FUNCTION_BLOCK FB_TouchProbe EXTENDS FB_Xfc
VAR
  _Ctrl             : REFERENCE TO ARRAY[1..MAX_TOUCH_PROBE] OF ST_CTRL_TOUCH_PROBE;
  _State            : REFERENCE TO ARRAY[1..MAX_TOUCH_PROBE] OF ST_STATE_TOUCH_PROBE;

  _Input            : POINTER TO ARRAY[1..MAX_TOUCH_PROBE] OF ST_MTI_Input;
  _InputState       : POINTER TO ARRAY[1..MAX_TOUCH_PROBE] OF ST_MTI_STATUS;

  _Index            : UDINT;
  _AxisId           : UDINT;
  _AxisIndex        : UDINT;

  _CtrlLocal        : ST_CTRL_TOUCH_PROBE;  // control data is copied to local on start of function
  _McDirection      : Tc2_MC2.MC_Direction;

  _eStateProgress   : E_PROGRESS;
  _eResult          : E_PROGRESS;

  _rtrigEnable      : Tc2_Standard.R_TRIG;
  _TrigCount        : UDINT;

  _CurrentTime      : ULINT;
  _CurrentTimeShort : UDINT;
  _LatchTime        : UDINT;
  _LatchState       : Bool;

  _bError           : BOOL;
  _stMsg            : ST_Message;
  _MessageLevel     : E_MessageType;
END_VAR

PROPERTY Ctrl : REFERENCE TO ARRAY [1..MAX_TOUCH_PROBE] OF ST_CTRL_TOUCH_PROBE
SET
_Ctrl REF= Ctrl;
END_SET
END_PROPERTY

METHOD Cycle : BOOL
VAR_INPUT
END_VAR
//-----------------------------------------------------------------------------
//-----------------------------------------------------------------------------
//  Check Enable
//-----------------------------------------------------------------------------
IF NOT _Ctrl[_Index].Enable
THEN
  // clear function state if not enabled
  _eStateProgress                   := E_PROGRESS.PROGRESS_INVALID;
  _LatchState                       := FALSE;
  _State[_Index].State              := TO_UINT(_eStateProgress);
END_IF
//-----------------------------------------------------------------------------
//-----------------------------------------------------------------------------
//  set message device
//-----------------------------------------------------------------------------
_eDeviceFunction                    := e_Device.XfcTouchProbe + _Index;
//-----------------------------------------------------------------------------
//-----------------------------------------------------------------------------
//  rising trigger react to enable command
//-----------------------------------------------------------------------------
_rtrigEnable(CLK                    := _Ctrl[_Index].Enable);
//-----------------------------------------------------------------------------
//-----------------------------------------------------------------------------
//  main state machine
//-----------------------------------------------------------------------------
CASE _eStateProgress
OF
  E_PROGRESS.PROGRESS_INVALID:      // check input data
    IF _rtrigEnable.Q
    THEN
      _State[_Index].State          := TO_UINT(E_PROGRESS.PROGRESS_BUSY);
      _State[_Index].LatchPositive  := 0.0;
      _State[_Index].LatchNegative  := 0.0;

      _bError                       := FALSE;
      _eStateProgress               := E_PROGRESS.PROGRESS_INIT;

      _CtrlLocal                    := _Ctrl[_Index];   // copy control data to local, you may write new data onto struct as long as .Enable stays TRUE
      _CurrentTime                  := Tc2_EtherCAT.F_GetCurDcTickTime64();
      _CurrentTimeShort             := TO_UDINT(_CurrentTime AND 16#FFFFFFFF);

      _AxisId                       := _CtrlLocal.AxisId;   // TwinCAT NC AxisId
      _AxisIndex                    := GetIndex(_AxisId);   // corresponding index in axis array

      _stMsg.iErrorNumber           := 0;

      IF NOT (_AxisIndex > 0) OR NOT (_AxisId > 0)
      THEN
        _bError                     := TRUE;
        _stMsg.iErrorNumber         := 1;
        _stMsg.sText                := 'AxisId Invalid ';
        _eStateProgress             := E_PROGRESS.PROGRESS_STILL_WORKING;
      END_IF

      IF NOT (_CtrlLocal.Direction = MC_Positive_Direction) OR 
         NOT (_CtrlLocal.Direction = MC_Negative_Direction)
      THEN
        _bError                     := TRUE;
        _stMsg.iErrorNumber         := 2;
        _stMsg.sText                := 'Direction Invalid ';
        _eStateProgress             := E_PROGRESS.PROGRESS_STILL_WORKING;
      END_IF

      IF NOT IsFinite(F_LReal(_CtrlLocal.PositionStart))
      THEN
        _bError                     := TRUE;
        _stMsg.iErrorNumber         := 3;
        _stMsg.sText                := 'PositionStart not finite ';
        _eStateProgress             := E_PROGRESS.PROGRESS_STILL_WORKING;
      END_IF

      IF NOT IsFinite(F_LReal(_CtrlLocal.PositionEnd))
      THEN
        _bError                     := TRUE;
        _stMsg.iErrorNumber         := 4;
        _stMsg.sText                := 'PositionEnd not finite ';
        _eStateProgress             := E_PROGRESS.PROGRESS_STILL_WORKING;
      END_IF
    END_IF

  E_PROGRESS.PROGRESS_INIT:
      _eDeviceAxis                  := e_Device.XfcAxis + (_CtrlLocal.AxisId);
      _eStateProgress               := E_PROGRESS.PROGRESS_BUSY;

      IF (_MessageLevel = E_MessageType.eMessageVerbose)
      THEN
        _stMsg.eType                := E_MessageType.eMessageVerbose;
        _stMsg.eDevice              := _eDeviceFunction;
        _stMsg.eSubdevice           := e_Subdevice.XfcTouchProbe;
        _stMsg.iErrorNumber         := _eDeviceAxis;
        _stMsg.sText                := concat(TO_STRING(_eStateProgress), ': ');
        _stMsg.sText                := concat(_stMsg.sText, TO_STRING(e_Device.XfcAxis));
        _stMsg.sText                := concat(_stMsg.sText, '_ID_');
        _stMsg.sText                := concat(_stMsg.sText, TO_STRING(_AxisId));

        f_MessageSet(_stMsg);
      END_IF
END_CASE
//-----------------------------------------------------------------------------
//-----------------------------------------------------------------------------
CASE _eStateProgress
OF
  E_PROGRESS.PROGRESS_BUSY:
    _McDirection                    := _CtrlLocal.Direction;
    CASE _McDirection
    OF
      MC_Positive_Direction:
        IF (_ItfAxis[_AxisIndex].Position >= _CtrlLocal.PositionStart)
        THEN
          _eResult                  := PositionAtTime(FALSE, _CtrlLocal.AxisId, 0, _MessageLevel);
          _eStateProgress           := E_PROGRESS.PROGRESS_PREPARE;
        END_IF

      MC_Negative_Direction:
        IF (_ItfAxis[_AxisIndex].Position <= _CtrlLocal.PositionStart)
        THEN
          _eResult                  := PositionAtTime(FALSE, _CtrlLocal.AxisId, 0, _MessageLevel);
          _eStateProgress           := E_PROGRESS.PROGRESS_PREPARE;
        END_IF
    END_CASE
END_CASE
//-----------------------------------------------------------------------------
//-----------------------------------------------------------------------------
CASE _eStateProgress
OF
  E_PROGRESS.PROGRESS_PREPARE:
    CASE _McDirection
    OF
      MC_Positive_Direction:
        IF (_ItfAxis[_AxisIndex].Position > _CtrlLocal.PositionEnd)
        THEN
          _bError                   := TRUE;
          _stMsg.iErrorNumber       := 5;
          _stMsg.sText              := 'PositionEnd reached, no rising trigger ';
          _eStateProgress           := E_PROGRESS.PROGRESS_STILL_WORKING;
    
        ELSIF (_Input^[_Index].EventState) OR
              (_Input^[_Index].EventTime > _CurrentTimeShort)
        THEN
          _LatchState               := _Input^[_Index].EventState;
          _LatchTime                := _Input^[_Index].EventTime;
    
          IF (_MessageLevel = E_MessageType.eMessageVerbose)
          THEN
            _stMsg.eType            := E_MessageType.eMessageVerbose;
            _stMsg.eDevice          := _eDeviceFunction;
            _stMsg.eSubdevice       := e_Subdevice.XfcTouchProbe;
            _stMsg.iErrorNumber     := _LatchTime;
            _stMsg.sText            := concat(TO_STRING(_eStateProgress), ': ');
            _stMsg.sText            := concat(_stMsg.sText, TO_STRING(e_Device.XfcAxis));
    
            f_MessageSet(_stMsg);
          END_IF
          _eStateProgress           := E_PROGRESS.PROGRESS_STARTUP;
        END_IF

      MC_Negative_Direction:
        IF (_ItfAxis[_AxisIndex].Position < _CtrlLocal.PositionEnd)
        THEN
          _bError                   := TRUE;
          _stMsg.iErrorNumber       := 5;
          _stMsg.sText              := 'PositionEnd reached, no rising trigger ';
          _eStateProgress           := E_PROGRESS.PROGRESS_STILL_WORKING;
    
        ELSIF (_Input^[_Index].EventState) OR
              (_Input^[_Index].EventTime > _CurrentTimeShort)
        THEN
          _LatchState               := _Input^[_Index].EventState;
          _LatchTime                := _Input^[_Index].EventTime;
    
          IF (_MessageLevel = E_MessageType.eMessageVerbose)
          THEN
            _stMsg.eType            := E_MessageType.eMessageVerbose;
            _stMsg.eDevice          := _eDeviceFunction;
            _stMsg.eSubdevice       := e_Subdevice.XfcTouchProbe;
            _stMsg.iErrorNumber     := _LatchTime;
            _stMsg.sText            := concat(TO_STRING(_eStateProgress), ': ');
            _stMsg.sText            := concat(_stMsg.sText, TO_STRING(e_Device.XfcAxis));
    
            f_MessageSet(_stMsg);
          END_IF
          _eStateProgress           := E_PROGRESS.PROGRESS_STARTUP;
        END_IF
    END_CASE
END_CASE
//-----------------------------------------------------------------------------
//-----------------------------------------------------------------------------
CASE _eStateProgress
OF
  E_PROGRESS.PROGRESS_STARTUP:
    _eResult                        := PositionAtTime(TRUE, _CtrlLocal.AxisId, _LatchTime, _MessageLevel);

    IF (_eResult = E_PROGRESS.PROGRESS_ERROR)
    THEN
      _bError                       := TRUE;
      _stMsg.iErrorNumber           := 7;
      _stMsg.sText                  := 'PositionAtTime LatchPositive ';
      _eStateProgress               := E_PROGRESS.PROGRESS_STILL_WORKING;
      _eResult                      := PositionAtTime(FALSE, _CtrlLocal.AxisId, 0, _MessageLevel);

    ELSIF (_eResult = E_PROGRESS.PROGRESS_DONE)
    THEN
      _State[_Index].LatchPositive  := _XfcRecordedPosition[_AxisIndex];

      _CurrentTime                  := Tc2_EtherCAT.F_GetCurDcTickTime64();
      _CurrentTimeShort             := TO_UDINT(_CurrentTime AND 16#FFFFFFFF);

      IF (_MessageLevel = E_MessageType.eMessageVerbose)
      THEN
        _stMsg.eType                := E_MessageType.eMessageVerbose;
        _stMsg.eDevice              := _eDeviceFunction;
        _stMsg.eSubdevice           := e_Subdevice.XfcTouchProbe;
        _stMsg.iErrorNumber         := _LatchTime;
        _stMsg.sText                := concat(TO_STRING(_eStateProgress), ': ');
        _stMsg.sText                := concat(_stMsg.sText, TO_STRING(_XfcRecordedPosition[_AxisIndex]));

        f_MessageSet(_stMsg);
      END_IF
      _eStateProgress               := E_PROGRESS.PROGRESS_CHECK;
      _eResult                      := PositionAtTime(FALSE, _CtrlLocal.AxisId, 0, _MessageLevel);
    END_IF
END_CASE
//-----------------------------------------------------------------------------
//-----------------------------------------------------------------------------
CASE _eStateProgress
OF
  E_PROGRESS.PROGRESS_CHECK:
    CASE _McDirection
    OF
      MC_Positive_Direction:
        IF (_ItfAxis[_AxisIndex].Position > _CtrlLocal.PositionEnd)
        THEN
          _bError                   := TRUE;
          _stMsg.iErrorNumber       := 6;
          _stMsg.sText              := concat('PositionEnd reached, no falling trigger :', TO_STRING(_ItfAxis[_AxisIndex].Position));
          _eStateProgress           := E_PROGRESS.PROGRESS_STILL_WORKING;
    
        ELSIF NOT (_Input^[_Index].EventState) OR
              (_Input^[_Index].EventTime > _LatchTime - 1_000)
        THEN
          _LatchState               := _Input^[_Index].EventState;
          _LatchTime                := _Input^[_Index].EventTime;
    
          IF (_MessageLevel = E_MessageType.eMessageVerbose)
          THEN
            _stMsg.eType            := E_MessageType.eMessageVerbose;
            _stMsg.eDevice          := _eDeviceFunction;
            _stMsg.eSubdevice       := e_Subdevice.XfcTouchProbe;
            _stMsg.iErrorNumber     := _LatchTime;
            _stMsg.sText            := concat(TO_STRING(_eStateProgress), ': ');
            _stMsg.sText            := concat(_stMsg.sText, TO_STRING(e_Device.XfcAxis));
    
            f_MessageSet(_stMsg);
          END_IF
          _eStateProgress           := E_PROGRESS.PROGRESS_OCCUPIED;
        END_IF

      MC_Negative_Direction:
        IF (_ItfAxis[_AxisIndex].Position < _CtrlLocal.PositionEnd)
        THEN
          _bError                   := TRUE;
          _stMsg.iErrorNumber       := 6;
          _stMsg.sText              := concat('PositionEnd reached, no falling trigger :', TO_STRING(_ItfAxis[_AxisIndex].Position));
          _eStateProgress           := E_PROGRESS.PROGRESS_STILL_WORKING;
    
        ELSIF NOT (_Input^[_Index].EventState) OR
              (_Input^[_Index].EventTime > _LatchTime - 1_000)
        THEN
          _LatchState               := _Input^[_Index].EventState;
          _LatchTime                := _Input^[_Index].EventTime;
    
          IF (_MessageLevel = E_MessageType.eMessageVerbose)
          THEN
            _stMsg.eType            := E_MessageType.eMessageVerbose;
            _stMsg.eDevice          := _eDeviceFunction;
            _stMsg.eSubdevice       := e_Subdevice.XfcTouchProbe;
            _stMsg.iErrorNumber     := _LatchTime;
            _stMsg.sText            := concat(TO_STRING(_eStateProgress), ': ');
            _stMsg.sText            := concat(_stMsg.sText, TO_STRING(e_Device.XfcAxis));
    
            f_MessageSet(_stMsg);
          END_IF
          _eStateProgress           := E_PROGRESS.PROGRESS_OCCUPIED;
        END_IF
    END_CASE
END_CASE
//-----------------------------------------------------------------------------
//-----------------------------------------------------------------------------
CASE _eStateProgress
OF
  E_PROGRESS.PROGRESS_OCCUPIED:
    _eResult                        := PositionAtTime(TRUE, _CtrlLocal.AxisId, _LatchTime, _MessageLevel);

    IF (_eResult = E_PROGRESS.PROGRESS_ERROR)
    THEN
      _bError                       := TRUE;
      _stMsg.iErrorNumber           := 8;
      _stMsg.sText                  := 'PositionAtTime LatchNegative: ';
      _eStateProgress               := E_PROGRESS.PROGRESS_STILL_WORKING;
      _eResult                      := PositionAtTime(FALSE, _CtrlLocal.AxisId, 0, _MessageLevel);

    ELSIF (_eResult = E_PROGRESS.PROGRESS_DONE)
    THEN
      _State[_Index].LatchNegative  := _XfcRecordedPosition[_AxisIndex];

      IF (_MessageLevel = E_MessageType.eMessageVerbose)
      THEN
        _stMsg.eType                := E_MessageType.eMessageVerbose;
        _stMsg.eDevice              := _eDeviceFunction;
        _stMsg.eSubdevice           := e_Subdevice.XfcTouchProbe;
        _stMsg.iErrorNumber         := _LatchTime;
        _stMsg.sText                := concat(TO_STRING(_eStateProgress), ': ');
        _stMsg.sText                := concat(_stMsg.sText, TO_STRING(_XfcRecordedPosition[_AxisIndex]));

        f_MessageSet(_stMsg);
      END_IF
      _eStateProgress               := E_PROGRESS.PROGRESS_WORKING;
      _eResult                      := PositionAtTime(FALSE, _CtrlLocal.AxisId, 0, _MessageLevel);
    END_IF
END_CASE
//-----------------------------------------------------------------------------
//-----------------------------------------------------------------------------
CASE _eStateProgress
OF
  E_PROGRESS.PROGRESS_WORKING:
    _eStateProgress                 := E_PROGRESS.PROGRESS_STILL_WORKING;
END_CASE
//-----------------------------------------------------------------------------
//-----------------------------------------------------------------------------
CASE _eStateProgress
OF
  E_PROGRESS.PROGRESS_STILL_WORKING:
    IF NOT _bError
    THEN
      _eStateProgress               := E_PROGRESS.PROGRESS_DONE;

      IF (_MessageLevel > E_MessageType.eMessageWarning)
      THEN
        _stMsg.eType                := E_MessageType.eMessageInfo;
        _stMsg.eDevice              := _eDeviceFunction;
        _stMsg.eSubdevice           := e_Subdevice.XfcTouchProbe;
        _stMsg.iErrorNumber         := _eDeviceAxis;
        _stMsg.sText                := concat(TO_STRING(_eStateProgress), ': ');
        _stMsg.sText                := concat(_stMsg.sText, TO_STRING(e_Device.XfcAxis));
        _stMsg.sText                := concat(_stMsg.sText, '_ID_');
        _stMsg.sText                := concat(_stMsg.sText, TO_STRING(_AxisId));

        f_MessageSet(_stMsg);
      END_IF
      _State[_Index].State          := TO_UINT(_eStateProgress);
    ELSE
      _eStateProgress               := E_PROGRESS.PROGRESS_ERROR;

      _stMsg.eType                  := E_MessageType.eMessageError;
      _stMsg.eDevice                := _eDeviceFunction;
      _stMsg.eSubdevice             := e_Subdevice.XfcTouchProbe;
      _stMsg.sText                  := concat(_stMsg.sText, TO_STRING(_eStateProgress));
      _stMsg.sText                  := concat(_stMsg.sText, ': ');
      _stMsg.sText                  := concat(_stMsg.sText, TO_STRING(e_Device.XfcAxis));
      _stMsg.sText                  := concat(_stMsg.sText, '_ID_');
      _stMsg.sText                  := concat(_stMsg.sText, TO_STRING(_AxisId));

      f_MessageSet(_stMsg);
      _State[_Index].State          := TO_UINT(_eStateProgress) + TO_UINT(_stMsg.iErrorNumber);
    END_IF
END_CASE
END_METHOD

PROPERTY Index : udint
GET
Index := _Index;
END_GET
SET
_Index := Index;
END_SET
END_PROPERTY

PROPERTY Input : pointer TO ARRAY [1..MAX_TOUCH_PROBE] OF ST_MTI_Input
SET
_Input := Input;
END_SET
END_PROPERTY

PROPERTY InputState : pointer TO ARRAY [1..MAX_TOUCH_PROBE] OF ST_MTI_STATUS
SET
_InputState := InputState;
END_SET
END_PROPERTY

PROPERTY MessageLevel : e_messagetype
GET
MessageLevel := _MessageLevel;
END_GET
SET
_MessageLevel := MessageLevel;
END_SET
END_PROPERTY

PROPERTY State :  REFERENCE TO ARRAY[1..MAX_TOUCH_PROBE] OF ST_STATE_TOUCH_PROBE;
SET
_State REF= State;
END_SET
END_PROPERTY

END_FUNCTION_BLOCK

(* stored: Version 1.1.0.1, ProductVersion 3.1.4026.18
   POU FB_TouchProbe: Id {379ba5cf-2e9d-498d-a8bf-d202d33bef2a}, SpecialFunc None
   Property Ctrl: Id {54fe8f3f-9445-437a-89b9-2c201fda5e98}
   Set Set: Id {dc10eecf-2bd5-4358-a169-ae96d39aa8b6}
   Method Cycle: Id {211e6416-a5ad-4ea8-a51c-fe35825bea80}
   Property Index: Id {2ad14ec0-74ba-4dc0-be2c-769aec1b401e}
   Get Get: Id {8c2feba7-3bfd-40e9-a587-1801df041bfa}
   Set Set: Id {181ace03-1c86-4c39-ab65-975367a2c1f7}
   Property Input: Id {54665186-7cbf-46fa-9f9f-24486f540965}
   Set Set: Id {1d54dd94-4fc9-4b7d-9746-161b9de3cd1c}
   Property InputState: Id {07bea674-c1e0-4819-b13a-24f0a7118b94}
   Set Set: Id {0e4bdfba-eb8f-444c-a9f7-a73c93697eba}
   Property MessageLevel: Id {d8c3388a-c45c-4862-8954-1cb7379f7dfe}
   Get Get: Id {66813ac6-89dd-48e1-89d1-07ff7edea78d}
   Set Set: Id {55ce8e29-5bc6-4e5a-829e-645018219a72}
   Property State: Id {2052e944-cac7-492a-8603-5996db9b1187}
   Set Set: Id {efd7f50d-8fb1-4fa7-bcf1-0c4997b1acb3} *)
